// TIA Portal V19 export
TYPE "Decoiler_Pers"
   STRUCT
      CoilDiamSensor : Struct
         Data : Struct
            AnalogicSensor_OffsetValue : Real := -3794.985;
            AnalogicSensor_OffsetValid : Bool := TRUE;
         END_STRUCT;
         Par : Struct
            AnalogicSensor_Enable : Bool := TRUE;
            AnalogicSensor_RangeLow : Real := 1000.0;
            AnalogicSensor_RangeHigh : Real := 3000.0;
            Diam_Min : Real := 500.0;
            Diam_Max : Real := 1800.0;
            EndCoil_Diam : Real;
            EndCoil_Timer : Time;
         END_STRUCT;
      END_STRUCT;
      Loop : Struct
         Par : Struct
            DelayRestartAfterMaxLoop : Time := T#500MS;
            DelayStopMaxLoop : Time := T#500MS;
            SensoAdjVel_PercentageMinus : LReal := 2.0;
            SensoAdjVel_PercentagePlus : LReal := 10.0;
            SensoAdjVel_PercentagePlusPlus : LReal := 30.0;
            SensoAdjVel_DelayPlusPlus : Time := T#10S;
         END_STRUCT;
      END_STRUCT;
      Feed : "SpeedMachine_Par";
      Coupling : Struct
         Engaged : Bool := TRUE;
      END_STRUCT;
      Jaws : Struct
         Par : Struct
            Pause : Time := T#10M;
            Duration : Time := T#5S;
            DiamEnable : Real := 550.0;
         END_STRUCT;
      END_STRUCT;
      PneumaticBracking : Struct
         DiameterChangeBrake : Real;
         BrakeLowSelected : Bool;
      END_STRUCT;
   END_STRUCT;
END_TYPE
